// Mitsubishi GX Works2 project: 2023-06-22 #1 생산자동화기능사 3번   PLC: Q03UDV
// 생산자동화기능사

// global labels: Global1
VAR_GLOBAL
  PB1 AT X0 : BOOL;
  PB2 AT X1 : BOOL;
  정지 AT X2 : BOOL;
  공급후진 AT X3 : BOOL;
  공급전진 AT X4 : BOOL;
  가공후진 AT X5 : BOOL;
  가공전진 AT X6 : BOOL;
  송출후진 AT X7 : BOOL;
  송출전진 AT X8 : BOOL;
  배출후진 AT X9 : BOOL;
  배출전진 AT X0A : BOOL;
  매거진 AT X0B : BOOL;
  금속센서 AT X0F : BOOL;
  PB3 AT X0C : BOOL;
  적색 AT Y20 : BOOL;
  황색 AT Y21 : BOOL;
  녹색 AT Y22 : BOOL;
  공급1 AT Y23 : BOOL;
  공급2 AT Y24 : BOOL;
  가공 AT Y25 : BOOL;
  드릴 AT Y26 : BOOL;
  송출 AT Y27 : BOOL;
  배출 AT Y28 : BOOL;
  컨베이어 AT Y29 : BOOL;
END_VAR

PROGRAM 테스트동작
VAR
  PHASE : INT;
END_VAR
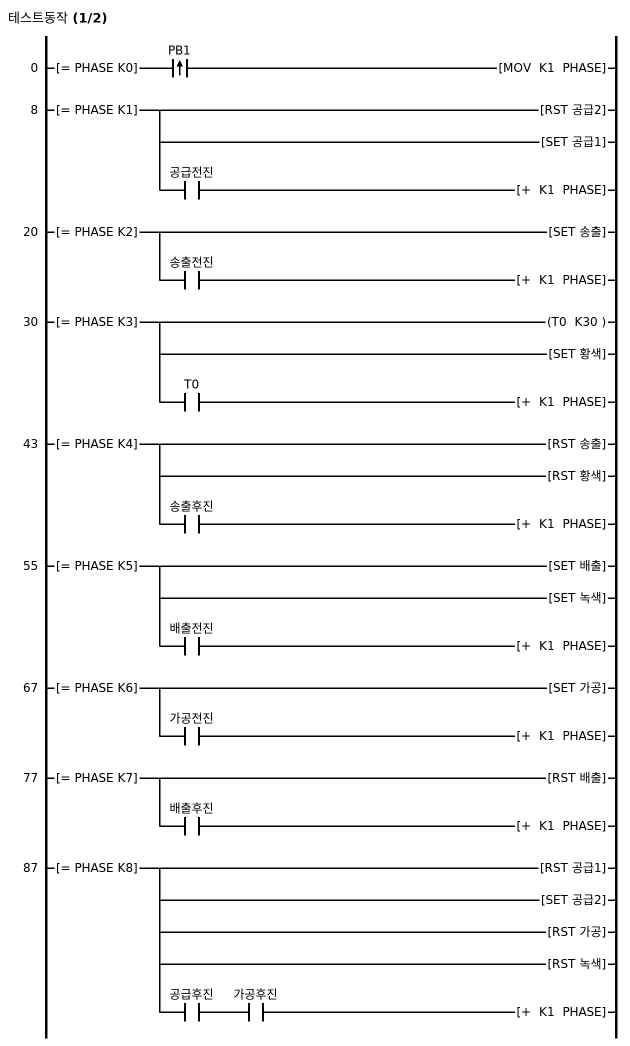
0     LD=     PHASE K0
      ANDP    PB1
      MOV     K1 PHASE
8     LD=     PHASE K1
      RST     공급2
      SET     공급1
      AND     공급전진
      +       K1 PHASE
20    LD=     PHASE K2
      SET     송출
      AND     송출전진
      +       K1 PHASE
30    LD=     PHASE K3
      OUT     T0 K30
      SET     황색
      AND     T0
      +       K1 PHASE
43    LD=     PHASE K4
      RST     송출
      RST     황색
      AND     송출후진
      +       K1 PHASE
55    LD=     PHASE K5
      SET     배출
      SET     녹색
      AND     배출전진
      +       K1 PHASE
67    LD=     PHASE K6
      SET     가공
      AND     가공전진
      +       K1 PHASE
77    LD=     PHASE K7
      RST     배출
      AND     배출후진
      +       K1 PHASE
87    LD=     PHASE K8
      RST     공급1
      SET     공급2
      RST     가공
      RST     녹색
      AND     공급후진
      AND     가공후진
      +       K1 PHASE
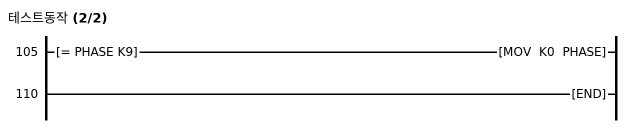
105   LD=     PHASE K9
      MOV     K0 PHASE
110   END
END_PROGRAM

PROGRAM 단속연속동작
VAR
  PHASE : INT;
  MODE : INT;
END_VAR
VAR CONSTANT
  단속 : INT;
  연속 : INT := 1;
END_VAR
VAR
  METAL : INT;
END_VAR
VAR CONSTANT
  금속 : INT := 1;
  비금속 : INT := 2;
END_VAR
VAR
  BLINK : ARRAY [0..7] OF BOOL;
  EMG : INT;
  PHASE1 : INT;
  황색1 : BOOL;
  녹색1 : BOOL;
  드릴1 : BOOL;
  컨베이어1 : BOOL;
END_VAR
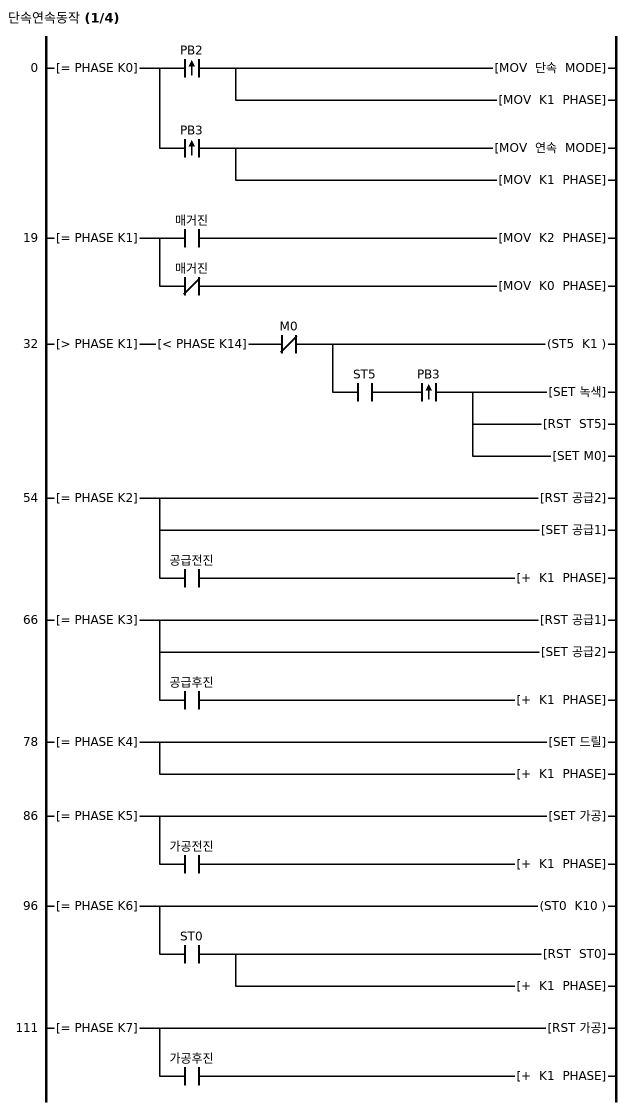
0     LD=     PHASE K0
      MPS
      ANDP    PB2
      MOV     단속 MODE
      MOV     K1 PHASE
      MPP
      ANDP    PB3
      MOV     연속 MODE
      MOV     K1 PHASE
19    LD=     PHASE K1
      MPS
      AND     매거진
      MOV     K2 PHASE
      MPP
      ANI     매거진
      MOV     K0 PHASE
32    LD>     PHASE K1
      AND<    PHASE K14
      ANI     M0
      OUT     ST5 K1
      AND     ST5
      ANDP    PB3
      SET     녹색
      RST     ST5
      SET     M0
54    LD=     PHASE K2
      RST     공급2
      SET     공급1
      AND     공급전진
      +       K1 PHASE
66    LD=     PHASE K3
      RST     공급1
      SET     공급2
      AND     공급후진
      +       K1 PHASE
78    LD=     PHASE K4
      SET     드릴
      +       K1 PHASE
86    LD=     PHASE K5
      SET     가공
      AND     가공전진
      +       K1 PHASE
96    LD=     PHASE K6
      OUT     ST0 K10
      AND     ST0
      RST     ST0
      +       K1 PHASE
111   LD=     PHASE K7
      RST     가공
      AND     가공후진
      +       K1 PHASE
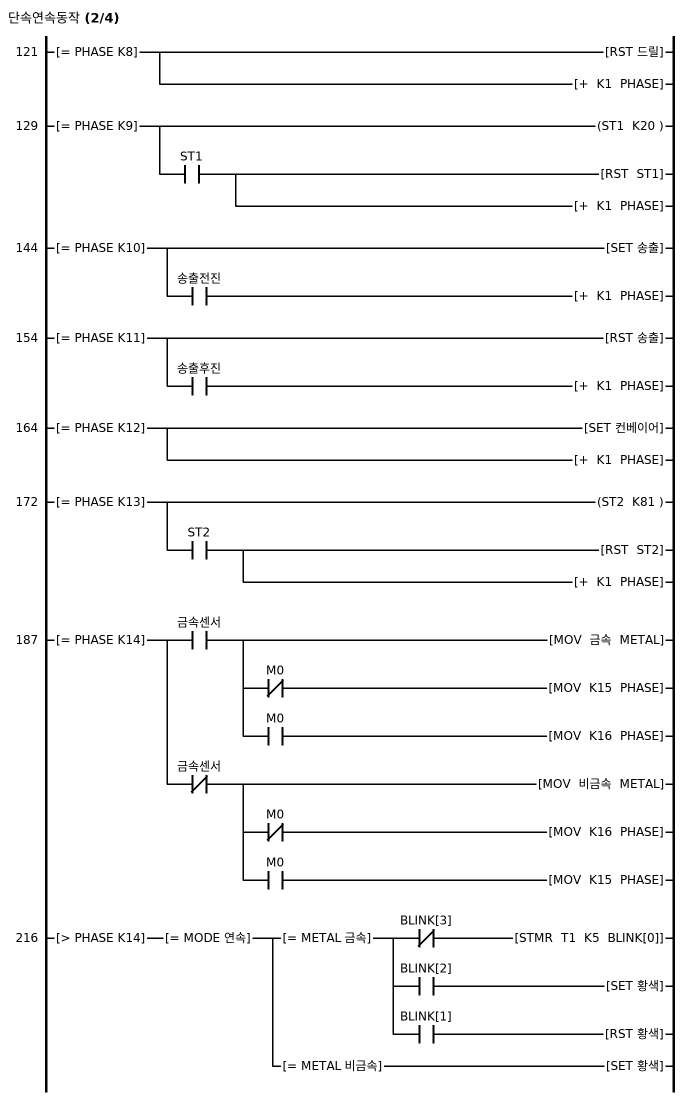
121   LD=     PHASE K8
      RST     드릴
      +       K1 PHASE
129   LD=     PHASE K9
      OUT     ST1 K20
      AND     ST1
      RST     ST1
      +       K1 PHASE
144   LD=     PHASE K10
      SET     송출
      AND     송출전진
      +       K1 PHASE
154   LD=     PHASE K11
      RST     송출
      AND     송출후진
      +       K1 PHASE
164   LD=     PHASE K12
      SET     컨베이어
      +       K1 PHASE
172   LD=     PHASE K13
      OUT     ST2 K81
      AND     ST2
      RST     ST2
      +       K1 PHASE
187   LD=     PHASE K14
      MPS
      AND     금속센서
      MOV     금속 METAL
      MPS
      ANI     M0
      MOV     K15 PHASE
      MPP
      AND     M0
      MOV     K16 PHASE
      MPP
      ANI     금속센서
      MOV     비금속 METAL
      MPS
      ANI     M0
      MOV     K16 PHASE
      MPP
      AND     M0
      MOV     K15 PHASE
216   LD>     PHASE K14
      AND=    MODE 연속
      MPS
      AND=    METAL 금속
      MPS
      ANI     BLINK[3]
      STMR    T1 K5 BLINK[0]
      MRD
      AND     BLINK[2]
      SET     황색
      MPP
      AND     BLINK[1]
      RST     황색
      MPP
      AND=    METAL 비금속
      SET     황색
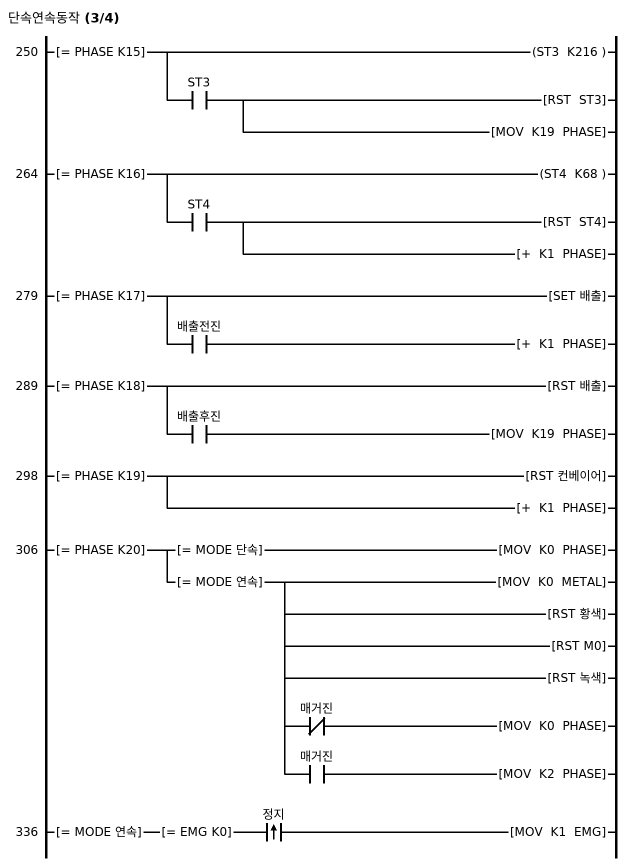
250   LD=     PHASE K15
      OUT     ST3 K216
      AND     ST3
      RST     ST3
      MOV     K19 PHASE
264   LD=     PHASE K16
      OUT     ST4 K68
      AND     ST4
      RST     ST4
      +       K1 PHASE
279   LD=     PHASE K17
      SET     배출
      AND     배출전진
      +       K1 PHASE
289   LD=     PHASE K18
      RST     배출
      AND     배출후진
      MOV     K19 PHASE
298   LD=     PHASE K19
      RST     컨베이어
      +       K1 PHASE
306   LD=     PHASE K20
      MPS
      AND=    MODE 단속
      MOV     K0 PHASE
      MPP
      AND=    MODE 연속
      MOV     K0 METAL
      RST     황색
      RST     M0
      RST     녹색
      MPS
      ANI     매거진
      MOV     K0 PHASE
      MPP
      AND     매거진
      MOV     K2 PHASE
336   LD=     MODE 연속
      AND=    EMG K0
      ANDP    정지
      MOV     K1 EMG
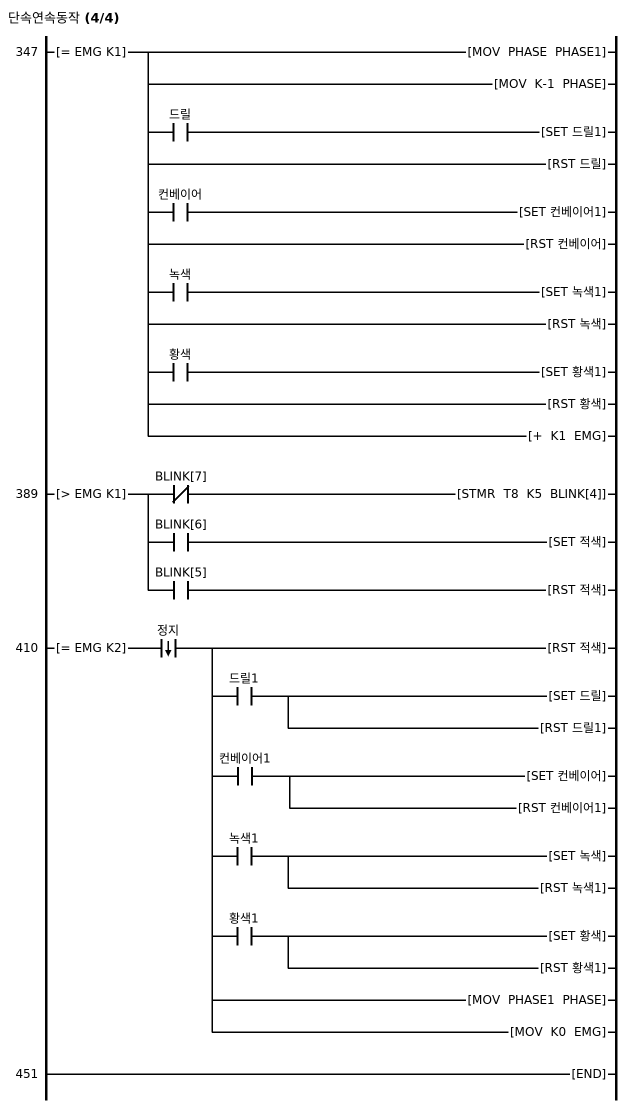
347   LD=     EMG K1
      MOV     PHASE PHASE1
      MOV     K-1 PHASE
      MPS
      AND     드릴
      SET     드릴1
      MPP
      RST     드릴
      MPS
      AND     컨베이어
      SET     컨베이어1
      MPP
      RST     컨베이어
      MPS
      AND     녹색
      SET     녹색1
      MPP
      RST     녹색
      MPS
      AND     황색
      SET     황색1
      MPP
      RST     황색
      +       K1 EMG
389   LD>     EMG K1
      MPS
      ANI     BLINK[7]
      STMR    T8 K5 BLINK[4]
      MRD
      AND     BLINK[6]
      SET     적색
      MPP
      AND     BLINK[5]
      RST     적색
410   LD=     EMG K2
      ANDF    정지
      RST     적색
      MPS
      AND     드릴1
      SET     드릴
      RST     드릴1
      MRD
      AND     컨베이어1
      SET     컨베이어
      RST     컨베이어1
      MRD
      AND     녹색1
      SET     녹색
      RST     녹색1
      MRD
      AND     황색1
      SET     황색
      RST     황색1
      MPP
      MOV     PHASE1 PHASE
      MOV     K0 EMG
451   END
END_PROGRAM
